// TIA Portal V20 export
FUNCTION_BLOCK "PartData"   // FB86, LAD
// stored: MemoryReserve 100, Namespace Unit1.Em5, SetENOAutomatically false
   VAR
      statQRCount { ExternalAccessible := 'False'; ExternalVisible := 'False'; ExternalWritable := 'False'} : DInt;
      statPulse { ExternalAccessible := 'False'; ExternalVisible := 'False'; ExternalWritable := 'False'} : Array[0..99] of Bool;
   END_VAR
   VAR_TEMP   // added for the SCL form of the ladder/FBD networks
      _w1 : Bool;
      _w2 : Bool;
      _w3 : Bool;
      _w4 : Bool;
      _w5 : Bool;
   END_VAR
BEGIN

REGION Network 1: QR ID Generate
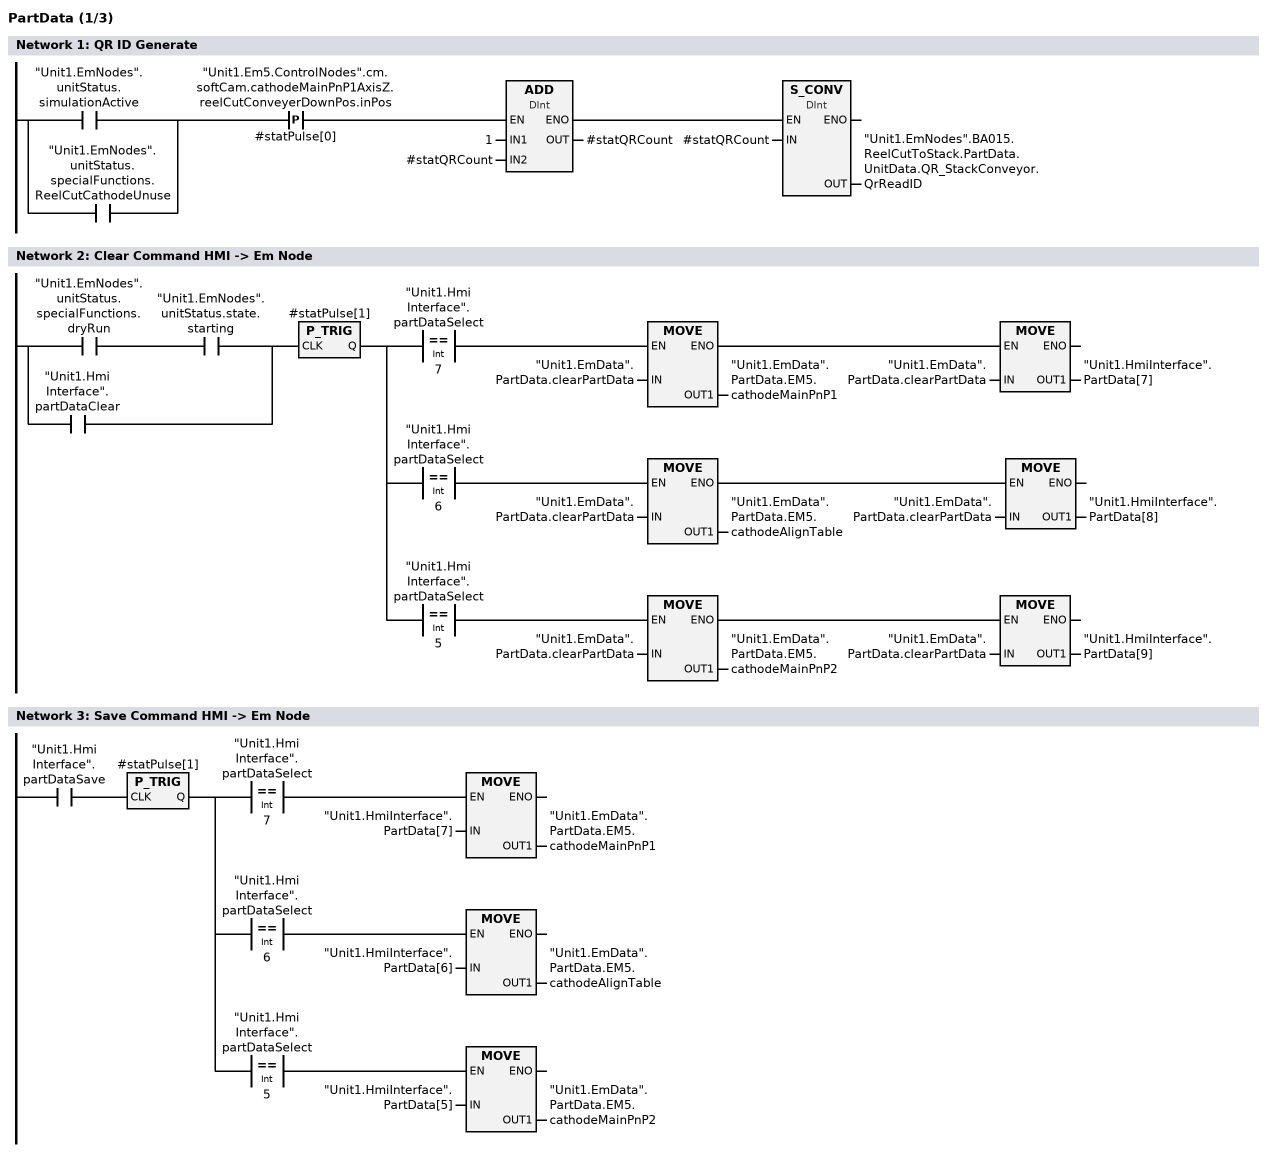
   RUNG wire#powerrail
      Contact( "Unit1.EmNodes".unitStatus.simulationActive )
      wire#w1
      P_Contact(operand := "Unit1.Em5.ControlNodes".cm.softCam.cathodeMainPnP1AxisZ.reelCutConveyerDownPos.inPos, bit := #statPulse[0])
      { S7_Templates := "SrcType := DInt" } Add(in1 := 1, in2 := #statQRCount, out => #statQRCount)
      { S7_Templates := "[src_type := DInt, dest_type := String]" } S_CONV(IN := #statQRCount, OUT => "Unit1.EmNodes".BA015.ReelCutToStack.PartData.UnitData.QR_StackConveyor.QrReadID)
   END_RUNG
   RUNG wire#powerrail
      Contact( "Unit1.EmNodes".unitStatus.specialFunctions.ReelCutCathodeUnuse )
   END_RUNG wire#w1
   // the same network as SCL:
   #_w1 := ("Unit1.EmNodes".unitStatus.simulationActive OR "Unit1.EmNodes".unitStatus.specialFunctions.ReelCutCathodeUnuse) AND "Unit1.Em5.ControlNodes".cm.softCam.cathodeMainPnP1AxisZ.reelCutConveyerDownPos.inPos AND NOT #statPulse[0];   // rising edge of "Unit1.Em5.ControlNodes".cm.softCam.cathodeMainPnP1AxisZ.reelCutConveyerDownPos.inPos
   #statPulse[0] := "Unit1.Em5.ControlNodes".cm.softCam.cathodeMainPnP1AxisZ.reelCutConveyerDownPos.inPos;
   IF #_w1 THEN
       #statQRCount := 1 + #statQRCount;
       S_CONV(IN := #statQRCount,
              OUT => "Unit1.EmNodes".BA015.ReelCutToStack.PartData.UnitData.QR_StackConveyor.QrReadID);
   END_IF;
END_REGION

REGION Network 2: Clear Command HMI -> Em Node
   RUNG wire#powerrail
      Contact( "Unit1.EmNodes".unitStatus.specialFunctions.dryRun )
      Contact( "Unit1.EmNodes".unitStatus.state.starting )
      wire#w1
      P_Trig( #statPulse[1] )
      wire#w2
      { S7_Templates := "SrcType := Int" } EQ_Contact(in1 := "Unit1.HmiInterface".partDataSelect, in2 := 7)
      Move(in := "Unit1.EmData".PartData.clearPartData, out1 => "Unit1.EmData".PartData.EM5.cathodeMainPnP1)
      Move(in := "Unit1.EmData".PartData.clearPartData, out1 => "Unit1.HmiInterface".PartData[7])
   END_RUNG
   RUNG wire#powerrail
      Contact( "Unit1.HmiInterface".partDataClear )
   END_RUNG wire#w1
   RUNG wire#w2
      { S7_Templates := "SrcType := Int" } EQ_Contact(in1 := "Unit1.HmiInterface".partDataSelect, in2 := 6)
      Move(in := "Unit1.EmData".PartData.clearPartData, out1 => "Unit1.EmData".PartData.EM5.cathodeAlignTable)
      Move(in := "Unit1.EmData".PartData.clearPartData, out1 => "Unit1.HmiInterface".PartData[8])
   END_RUNG
   RUNG wire#w2
      { S7_Templates := "SrcType := Int" } EQ_Contact(in1 := "Unit1.HmiInterface".partDataSelect, in2 := 5)
      Move(in := "Unit1.EmData".PartData.clearPartData, out1 => "Unit1.EmData".PartData.EM5.cathodeMainPnP2)
      Move(in := "Unit1.EmData".PartData.clearPartData, out1 => "Unit1.HmiInterface".PartData[9])
   END_RUNG
   // the same network as SCL:
   #_w1 := ("Unit1.EmNodes".unitStatus.specialFunctions.dryRun AND "Unit1.EmNodes".unitStatus.state.starting) OR "Unit1.HmiInterface".partDataClear;
   #_w2 := #_w1 AND NOT #statPulse[1];   // rising edge
   #statPulse[1] := #_w1;
   IF #_w2 AND ("Unit1.HmiInterface".partDataSelect = 7) THEN
       "Unit1.EmData".PartData.EM5.cathodeMainPnP1 := "Unit1.EmData".PartData.clearPartData;
       "Unit1.HmiInterface".PartData[7] := "Unit1.EmData".PartData.clearPartData;
   END_IF;
   IF #_w2 AND ("Unit1.HmiInterface".partDataSelect = 6) THEN
       "Unit1.EmData".PartData.EM5.cathodeAlignTable := "Unit1.EmData".PartData.clearPartData;
       "Unit1.HmiInterface".PartData[8] := "Unit1.EmData".PartData.clearPartData;
   END_IF;
   IF #_w2 AND ("Unit1.HmiInterface".partDataSelect = 5) THEN
       "Unit1.EmData".PartData.EM5.cathodeMainPnP2 := "Unit1.EmData".PartData.clearPartData;
       "Unit1.HmiInterface".PartData[9] := "Unit1.EmData".PartData.clearPartData;
   END_IF;
END_REGION

REGION Network 3: Save Command HMI -> Em Node
   RUNG wire#powerrail
      Contact( "Unit1.HmiInterface".partDataSave )
      P_Trig( #statPulse[1] )
      wire#w1
      { S7_Templates := "SrcType := Int" } EQ_Contact(in1 := "Unit1.HmiInterface".partDataSelect, in2 := 7)
      Move(in := "Unit1.HmiInterface".PartData[7], out1 => "Unit1.EmData".PartData.EM5.cathodeMainPnP1)
   END_RUNG
   RUNG wire#w1
      { S7_Templates := "SrcType := Int" } EQ_Contact(in1 := "Unit1.HmiInterface".partDataSelect, in2 := 6)
      Move(in := "Unit1.HmiInterface".PartData[6], out1 => "Unit1.EmData".PartData.EM5.cathodeAlignTable)
   END_RUNG
   RUNG wire#w1
      { S7_Templates := "SrcType := Int" } EQ_Contact(in1 := "Unit1.HmiInterface".partDataSelect, in2 := 5)
      Move(in := "Unit1.HmiInterface".PartData[5], out1 => "Unit1.EmData".PartData.EM5.cathodeMainPnP2)
   END_RUNG
   // the same network as SCL:
   #_w1 := "Unit1.HmiInterface".partDataSave AND NOT #statPulse[1];   // rising edge
   #statPulse[1] := "Unit1.HmiInterface".partDataSave;
   IF #_w1 AND ("Unit1.HmiInterface".partDataSelect = 7) THEN
       "Unit1.EmData".PartData.EM5.cathodeMainPnP1 := "Unit1.HmiInterface".PartData[7];
   END_IF;
   IF #_w1 AND ("Unit1.HmiInterface".partDataSelect = 6) THEN
       "Unit1.EmData".PartData.EM5.cathodeAlignTable := "Unit1.HmiInterface".PartData[6];
   END_IF;
   IF #_w1 AND ("Unit1.HmiInterface".partDataSelect = 5) THEN
       "Unit1.EmData".PartData.EM5.cathodeMainPnP2 := "Unit1.HmiInterface".PartData[5];
   END_IF;
END_REGION

REGION Network 4
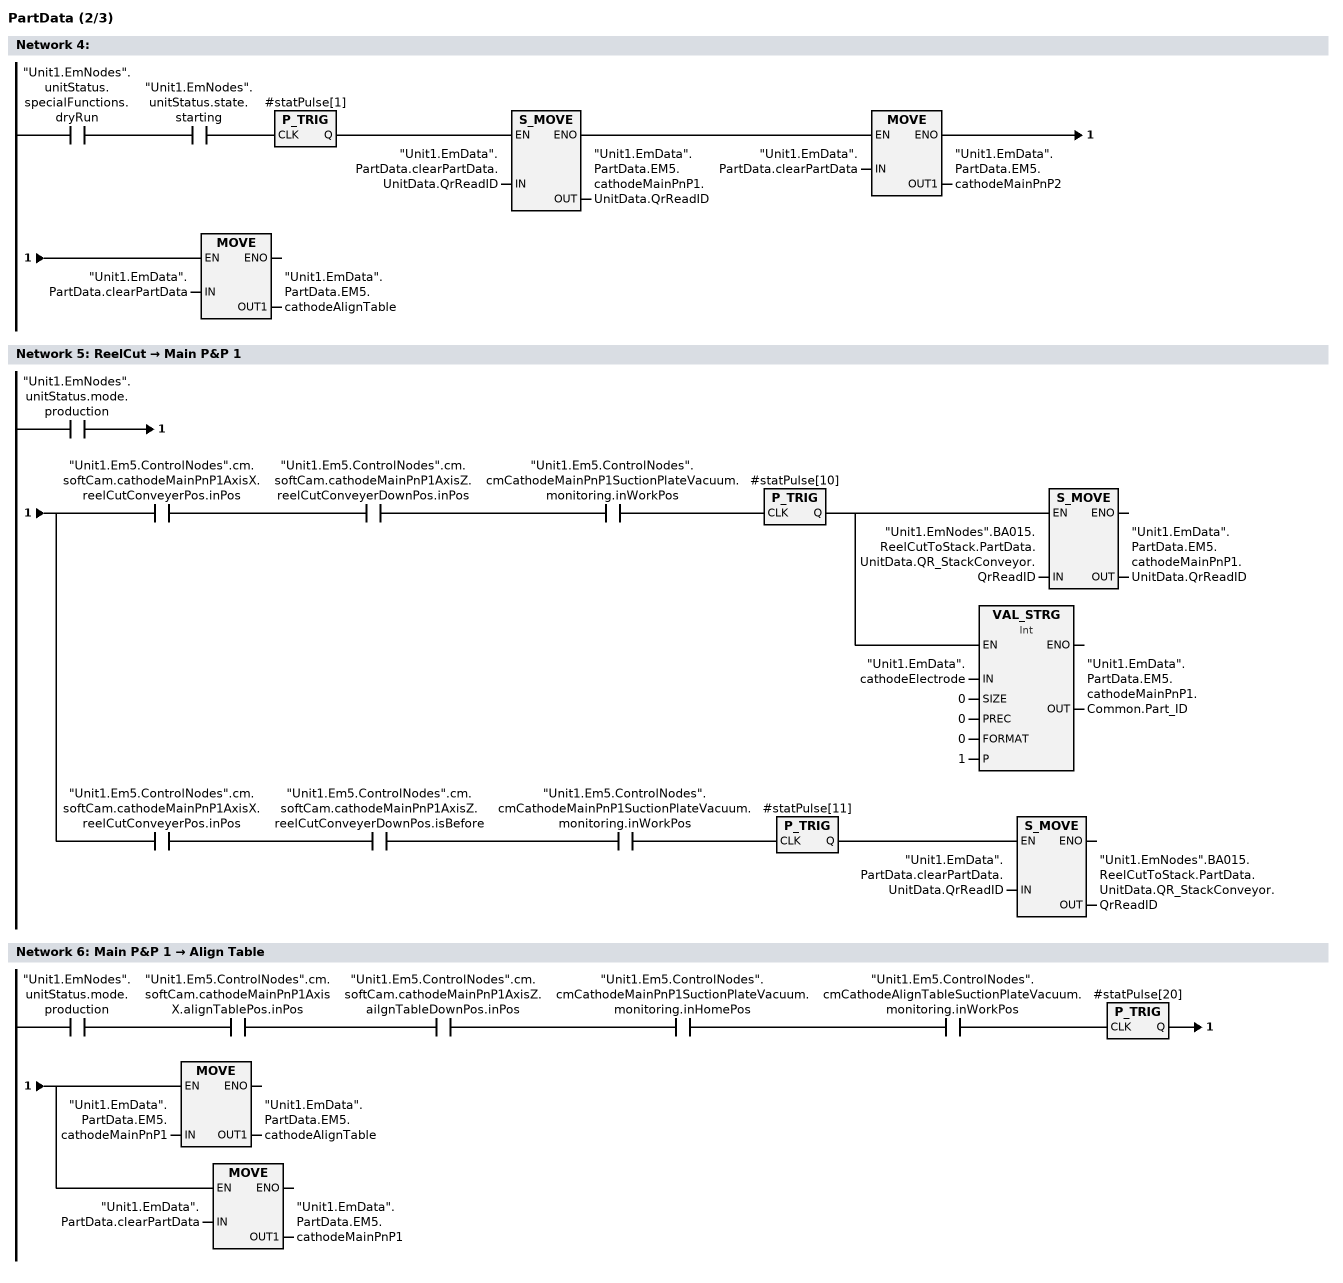
   RUNG wire#powerrail
      Contact( "Unit1.EmNodes".unitStatus.specialFunctions.dryRun )
      Contact( "Unit1.EmNodes".unitStatus.state.starting )
      P_Trig( #statPulse[1] )
      S_Move(in := "Unit1.EmData".PartData.clearPartData.UnitData.QrReadID, out => "Unit1.EmData".PartData.EM5.cathodeMainPnP1.UnitData.QrReadID)
      Move(in := "Unit1.EmData".PartData.clearPartData, out1 => "Unit1.EmData".PartData.EM5.cathodeMainPnP2)
      Move(in := "Unit1.EmData".PartData.clearPartData, out1 => "Unit1.EmData".PartData.EM5.cathodeAlignTable)
   END_RUNG
   // the same network as SCL:
   #_w1 := "Unit1.EmNodes".unitStatus.specialFunctions.dryRun AND "Unit1.EmNodes".unitStatus.state.starting;
   #_w2 := #_w1 AND NOT #statPulse[1];   // rising edge
   #statPulse[1] := #_w1;
   IF #_w2 THEN
       "Unit1.EmData".PartData.EM5.cathodeMainPnP1.UnitData.QrReadID := "Unit1.EmData".PartData.clearPartData.UnitData.QrReadID;
       "Unit1.EmData".PartData.EM5.cathodeMainPnP2 := "Unit1.EmData".PartData.clearPartData;
       "Unit1.EmData".PartData.EM5.cathodeAlignTable := "Unit1.EmData".PartData.clearPartData;
   END_IF;
END_REGION

REGION Network 5: ReelCut → Main P&P 1
   RUNG wire#powerrail
      Contact( "Unit1.EmNodes".unitStatus.mode.production )
      wire#w1
      Contact( "Unit1.Em5.ControlNodes".cm.softCam.cathodeMainPnP1AxisX.reelCutConveyerPos.inPos )
      Contact( "Unit1.Em5.ControlNodes".cm.softCam.cathodeMainPnP1AxisZ.reelCutConveyerDownPos.inPos )
      Contact( "Unit1.Em5.ControlNodes".cmCathodeMainPnP1SuctionPlateVacuum.monitoring.inWorkPos )
      P_Trig( #statPulse[10] )
      wire#w2
      S_Move(in := "Unit1.EmNodes".BA015.ReelCutToStack.PartData.UnitData.QR_StackConveyor.QrReadID, out => "Unit1.EmData".PartData.EM5.cathodeMainPnP1.UnitData.QrReadID)
   END_RUNG
   RUNG wire#w2
      { S7_Templates := "[value_type := Int, str_type := String]" } VAL_STRG(IN := "Unit1.EmData".cathodeElectrode, SIZE := 0, PREC := 0, FORMAT := 0, P := 1, OUT => "Unit1.EmData".PartData.EM5.cathodeMainPnP1.Common.Part_ID)
   END_RUNG
   RUNG wire#w1
      Contact( "Unit1.Em5.ControlNodes".cm.softCam.cathodeMainPnP1AxisX.reelCutConveyerPos.inPos )
      Contact( "Unit1.Em5.ControlNodes".cm.softCam.cathodeMainPnP1AxisZ.reelCutConveyerDownPos.isBefore )
      Contact( "Unit1.Em5.ControlNodes".cmCathodeMainPnP1SuctionPlateVacuum.monitoring.inWorkPos )
      P_Trig( #statPulse[11] )
      S_Move(in := "Unit1.EmData".PartData.clearPartData.UnitData.QrReadID, out => "Unit1.EmNodes".BA015.ReelCutToStack.PartData.UnitData.QR_StackConveyor.QrReadID)
   END_RUNG
   // the same network as SCL:
   #_w1 := "Unit1.EmNodes".unitStatus.mode.production AND "Unit1.Em5.ControlNodes".cm.softCam.cathodeMainPnP1AxisX.reelCutConveyerPos.inPos AND "Unit1.Em5.ControlNodes".cm.softCam.cathodeMainPnP1AxisZ.reelCutConveyerDownPos.inPos AND "Unit1.Em5.ControlNodes".cmCathodeMainPnP1SuctionPlateVacuum.monitoring.inWorkPos;
   #_w2 := #_w1 AND NOT #statPulse[10];   // rising edge
   #statPulse[10] := #_w1;
   IF #_w2 THEN
       "Unit1.EmData".PartData.EM5.cathodeMainPnP1.UnitData.QrReadID := "Unit1.EmNodes".BA015.ReelCutToStack.PartData.UnitData.QR_StackConveyor.QrReadID;
   END_IF;
   #_w3 := "Unit1.EmNodes".unitStatus.mode.production;
   IF #_w2 THEN
       VAL_STRG(IN := "Unit1.EmData".cathodeElectrode,
                SIZE := 0,
                PREC := 0,
                FORMAT := 0,
                P := 1,
                OUT => "Unit1.EmData".PartData.EM5.cathodeMainPnP1.Common.Part_ID);
   END_IF;
   #_w4 := #_w3 AND "Unit1.Em5.ControlNodes".cm.softCam.cathodeMainPnP1AxisX.reelCutConveyerPos.inPos AND "Unit1.Em5.ControlNodes".cm.softCam.cathodeMainPnP1AxisZ.reelCutConveyerDownPos.isBefore AND "Unit1.Em5.ControlNodes".cmCathodeMainPnP1SuctionPlateVacuum.monitoring.inWorkPos;
   #_w5 := #_w4 AND NOT #statPulse[11];   // rising edge
   #statPulse[11] := #_w4;
   IF #_w5 THEN
       "Unit1.EmNodes".BA015.ReelCutToStack.PartData.UnitData.QR_StackConveyor.QrReadID := "Unit1.EmData".PartData.clearPartData.UnitData.QrReadID;
   END_IF;
END_REGION

REGION Network 6: Main P&P 1 → Align Table
   RUNG wire#powerrail
      Contact( "Unit1.EmNodes".unitStatus.mode.production )
      Contact( "Unit1.Em5.ControlNodes".cm.softCam.cathodeMainPnP1AxisX.alignTablePos.inPos )
      Contact( "Unit1.Em5.ControlNodes".cm.softCam.cathodeMainPnP1AxisZ.ailgnTableDownPos.inPos )
      Contact( "Unit1.Em5.ControlNodes".cmCathodeMainPnP1SuctionPlateVacuum.monitoring.inHomePos )
      Contact( "Unit1.Em5.ControlNodes".cmCathodeAlignTableSuctionPlateVacuum.monitoring.inWorkPos )
      P_Trig( #statPulse[20] )
      wire#w1
      Move(in := "Unit1.EmData".PartData.EM5.cathodeMainPnP1, out1 => "Unit1.EmData".PartData.EM5.cathodeAlignTable)
   END_RUNG
   RUNG wire#w1
      Move(in := "Unit1.EmData".PartData.clearPartData, out1 => "Unit1.EmData".PartData.EM5.cathodeMainPnP1)
   END_RUNG
   // the same network as SCL:
   #_w1 := "Unit1.EmNodes".unitStatus.mode.production AND "Unit1.Em5.ControlNodes".cm.softCam.cathodeMainPnP1AxisX.alignTablePos.inPos AND "Unit1.Em5.ControlNodes".cm.softCam.cathodeMainPnP1AxisZ.ailgnTableDownPos.inPos AND "Unit1.Em5.ControlNodes".cmCathodeMainPnP1SuctionPlateVacuum.monitoring.inHomePos AND "Unit1.Em5.ControlNodes".cmCathodeAlignTableSuctionPlateVacuum.monitoring.inWorkPos;
   #_w2 := #_w1 AND NOT #statPulse[20];   // rising edge
   #statPulse[20] := #_w1;
   IF #_w2 THEN
       "Unit1.EmData".PartData.EM5.cathodeAlignTable := "Unit1.EmData".PartData.EM5.cathodeMainPnP1;
       "Unit1.EmData".PartData.EM5.cathodeMainPnP1 := "Unit1.EmData".PartData.clearPartData;
   END_IF;
END_REGION

REGION Network 7: Align Table → Main P&P 2
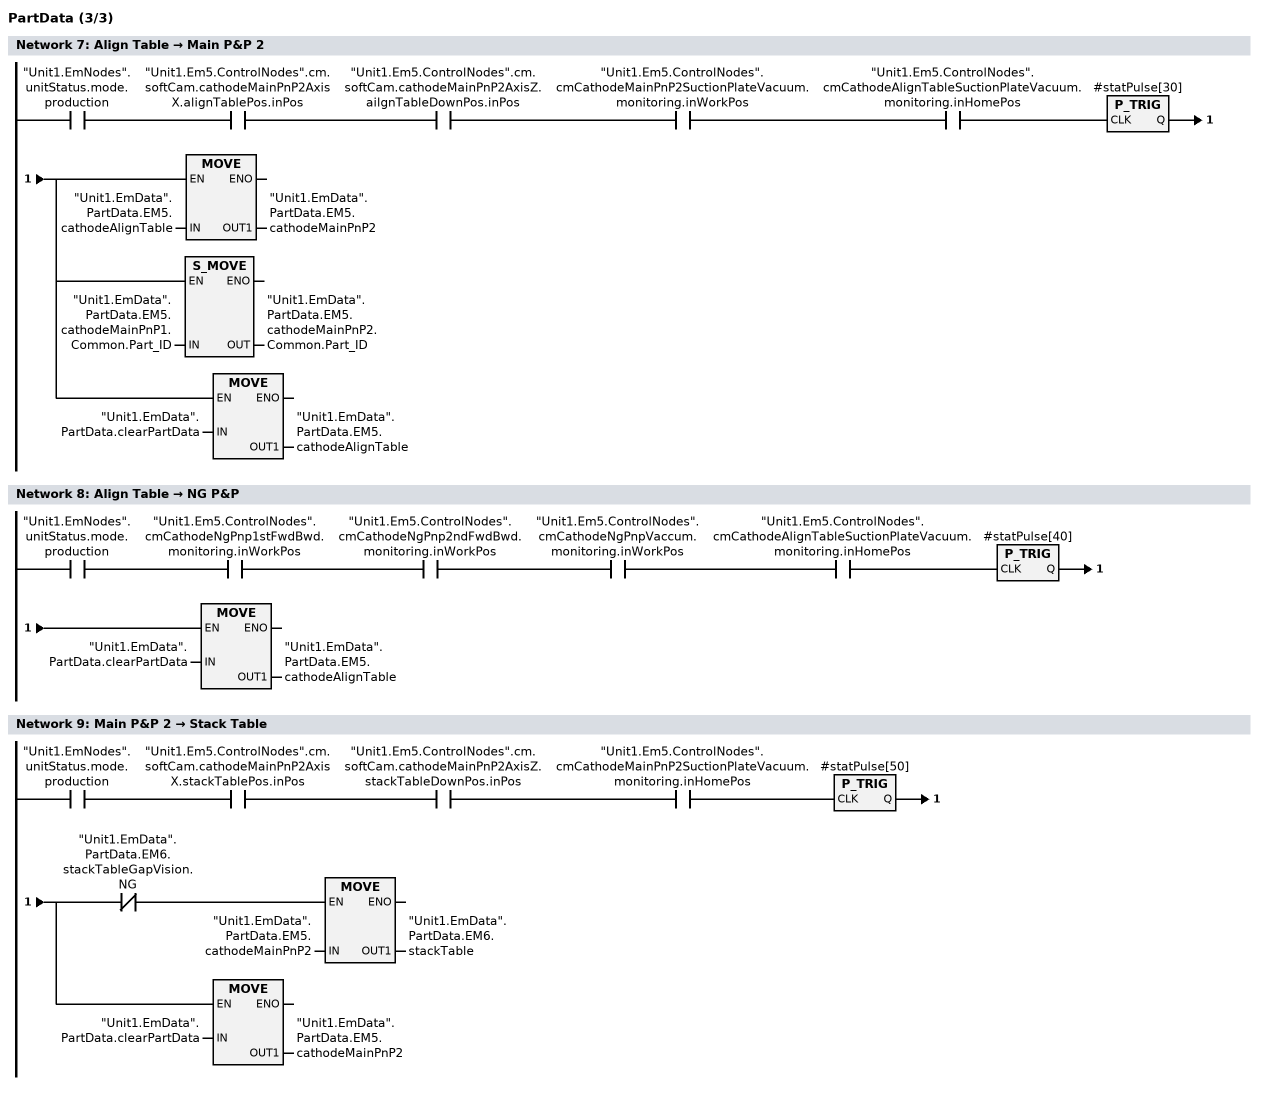
   RUNG wire#powerrail
      Contact( "Unit1.EmNodes".unitStatus.mode.production )
      Contact( "Unit1.Em5.ControlNodes".cm.softCam.cathodeMainPnP2AxisX.alignTablePos.inPos )
      Contact( "Unit1.Em5.ControlNodes".cm.softCam.cathodeMainPnP2AxisZ.ailgnTableDownPos.inPos )
      Contact( "Unit1.Em5.ControlNodes".cmCathodeMainPnP2SuctionPlateVacuum.monitoring.inWorkPos )
      Contact( "Unit1.Em5.ControlNodes".cmCathodeAlignTableSuctionPlateVacuum.monitoring.inHomePos )
      P_Trig( #statPulse[30] )
      wire#w1
      Move(in := "Unit1.EmData".PartData.EM5.cathodeAlignTable, out1 => "Unit1.EmData".PartData.EM5.cathodeMainPnP2)
   END_RUNG
   RUNG wire#w1
      S_Move(in := "Unit1.EmData".PartData.EM5.cathodeMainPnP1.Common.Part_ID, out => "Unit1.EmData".PartData.EM5.cathodeMainPnP2.Common.Part_ID)
   END_RUNG
   RUNG wire#w1
      Move(in := "Unit1.EmData".PartData.clearPartData, out1 => "Unit1.EmData".PartData.EM5.cathodeAlignTable)
   END_RUNG
   // the same network as SCL:
   #_w1 := "Unit1.EmNodes".unitStatus.mode.production AND "Unit1.Em5.ControlNodes".cm.softCam.cathodeMainPnP2AxisX.alignTablePos.inPos AND "Unit1.Em5.ControlNodes".cm.softCam.cathodeMainPnP2AxisZ.ailgnTableDownPos.inPos AND "Unit1.Em5.ControlNodes".cmCathodeMainPnP2SuctionPlateVacuum.monitoring.inWorkPos AND "Unit1.Em5.ControlNodes".cmCathodeAlignTableSuctionPlateVacuum.monitoring.inHomePos;
   #_w2 := #_w1 AND NOT #statPulse[30];   // rising edge
   #statPulse[30] := #_w1;
   IF #_w2 THEN
       "Unit1.EmData".PartData.EM5.cathodeMainPnP2 := "Unit1.EmData".PartData.EM5.cathodeAlignTable;
       "Unit1.EmData".PartData.EM5.cathodeMainPnP2.Common.Part_ID := "Unit1.EmData".PartData.EM5.cathodeMainPnP1.Common.Part_ID;
       "Unit1.EmData".PartData.EM5.cathodeAlignTable := "Unit1.EmData".PartData.clearPartData;
   END_IF;
END_REGION

REGION Network 8: Align Table → NG P&P
   RUNG wire#powerrail
      Contact( "Unit1.EmNodes".unitStatus.mode.production )
      Contact( "Unit1.Em5.ControlNodes".cmCathodeNgPnp1stFwdBwd.monitoring.inWorkPos )
      Contact( "Unit1.Em5.ControlNodes".cmCathodeNgPnp2ndFwdBwd.monitoring.inWorkPos )
      Contact( "Unit1.Em5.ControlNodes".cmCathodeNgPnpVaccum.monitoring.inWorkPos )
      Contact( "Unit1.Em5.ControlNodes".cmCathodeAlignTableSuctionPlateVacuum.monitoring.inHomePos )
      P_Trig( #statPulse[40] )
      Move(in := "Unit1.EmData".PartData.clearPartData, out1 => "Unit1.EmData".PartData.EM5.cathodeAlignTable)
   END_RUNG
   // the same network as SCL:
   #_w1 := "Unit1.EmNodes".unitStatus.mode.production AND "Unit1.Em5.ControlNodes".cmCathodeNgPnp1stFwdBwd.monitoring.inWorkPos AND "Unit1.Em5.ControlNodes".cmCathodeNgPnp2ndFwdBwd.monitoring.inWorkPos AND "Unit1.Em5.ControlNodes".cmCathodeNgPnpVaccum.monitoring.inWorkPos AND "Unit1.Em5.ControlNodes".cmCathodeAlignTableSuctionPlateVacuum.monitoring.inHomePos;
   #_w2 := #_w1 AND NOT #statPulse[40];   // rising edge
   #statPulse[40] := #_w1;
   IF #_w2 THEN
       "Unit1.EmData".PartData.EM5.cathodeAlignTable := "Unit1.EmData".PartData.clearPartData;
   END_IF;
END_REGION

REGION Network 9: Main P&P 2 → Stack Table
   RUNG wire#powerrail
      Contact( "Unit1.EmNodes".unitStatus.mode.production )
      Contact( "Unit1.Em5.ControlNodes".cm.softCam.cathodeMainPnP2AxisX.stackTablePos.inPos )
      Contact( "Unit1.Em5.ControlNodes".cm.softCam.cathodeMainPnP2AxisZ.stackTableDownPos.inPos )
      Contact( "Unit1.Em5.ControlNodes".cmCathodeMainPnP2SuctionPlateVacuum.monitoring.inHomePos )
      P_Trig( #statPulse[50] )
      wire#w1
      I_Contact( "Unit1.EmData".PartData.EM6.stackTableGapVision.NG )
      Move(in := "Unit1.EmData".PartData.EM5.cathodeMainPnP2, out1 => "Unit1.EmData".PartData.EM6.stackTable)
   END_RUNG
   RUNG wire#w1
      Move(in := "Unit1.EmData".PartData.clearPartData, out1 => "Unit1.EmData".PartData.EM5.cathodeMainPnP2)
   END_RUNG
   // the same network as SCL:
   #_w1 := "Unit1.EmNodes".unitStatus.mode.production AND "Unit1.Em5.ControlNodes".cm.softCam.cathodeMainPnP2AxisX.stackTablePos.inPos AND "Unit1.Em5.ControlNodes".cm.softCam.cathodeMainPnP2AxisZ.stackTableDownPos.inPos AND "Unit1.Em5.ControlNodes".cmCathodeMainPnP2SuctionPlateVacuum.monitoring.inHomePos;
   #_w2 := #_w1 AND NOT #statPulse[50];   // rising edge
   #statPulse[50] := #_w1;
   IF #_w2 AND NOT "Unit1.EmData".PartData.EM6.stackTableGapVision.NG THEN
       "Unit1.EmData".PartData.EM6.stackTable := "Unit1.EmData".PartData.EM5.cathodeMainPnP2;
   END_IF;
   IF #_w2 THEN "Unit1.EmData".PartData.EM5.cathodeMainPnP2 := "Unit1.EmData".PartData.clearPartData; END_IF;
END_REGION
END_FUNCTION_BLOCK
